(* Schneider Machine Expert - Basic project resolucao, file version 2.7.0.0 *)
(* ProjectInformations: Name=Novo projeto *)

HARDWARE
  Cpu 0: TM221M16R/G
  ModuleExtensionObject 0: TM3DQ16TK
  EthernetConfiguration: NetworkName=M221, IpAllocationMode=FixedAddress, IpAddress=0.0.0.0, SubnetMask=0.0.0.0
  SerialLineConfiguration: Baud=Baud19200, Parity=ParityEven, DataBits=DataBits8, StopBits=StopBits1, PhysicalMedium=PhysicalMediumRs485, TransmissionMode=TransmissionModeModbusRtu, SlaveId=1, Addressing=SlaveAddressing
  MastTask: UsePeriodScanMode=false, PeriodScan=100
  FastTask: Period=255
  CpuBehavior: StartingMode=StartAsPreviousState, AutoSaveRamOnEeprom=true, WatchdogPeriod=250

SYMBOLS  (address, symbol, comment, settings)
  %M0       SIG_IN_BOT_P1
  %M1       SIG_IN_BOT_P2
  %M2       SIG_IN_SEN_A
  %M3       SIG_IN_SEN_B
  %M4       SIG_IN_SEN_C
  %M5       SIG_IN_SEN_D1
  %M6       SIG_IN_SEN_D2
  %M10      SIG_E1_E2E3
  %M11      SIG_E2_E4
  %M13      SIG_E4_E6
  %M15      SIG_E6_E8
  %M17      SIG_E8_E10
  %M20      SIG_OUT_M1
  %M21      SIG_OUT_M1_INV
  %M22      SIG_OUT_M2
  %M23      SIG_OUT_M2_INV
  %M24      SIG_OUT_M3
  %M25      SIG_OUT_M3_INV
  %M26      SIG_OUT_M4
  %M27      SIG_OUT_M4_INV
  %M28      SIG_OUT_ATU_V1
  %M30      SIG_CAR_I_C
  %M31      SIG_CAR_II_C
  %M40      SIG_E10_E12
  %X1       E1
  %X2       E2
  %X3       E3
  %X4       E4
  %X5       E5
  %X6       E6
  %X7       E7
  %X8       E8
  %X9       E9
  %X10      E10
  %TM0      FT_E6_E8  [Preset=2, Base=OneSecond]
  %TM2      FT_E10_E12  [Preset=5, Base=OneSecond]
  %I0.0     IN_BOT_P1
  %I0.1     IN_BOT_P2
  %I0.2     IN_SEN_A
  %I0.3     IN_SEN_B
  %I0.4     IN_SEN_C
  %I0.5     IN_SEN_D1
  %I0.6     IN_SEN_D2
  %Q0.0     OUT_M1
  %Q0.1     OUT_M1_INV
  %Q0.2     OUT_M2
  %Q0.3     OUT_M2_INV
  %Q0.4     OUT_M3
  %Q0.5     OUT_M3_INV
  %Q0.6     OUT_M4
  %Q0.7     OUT_M4_INV
  %Q1.0     OUT_ATU_V1

GRAFCET Grafcet POU
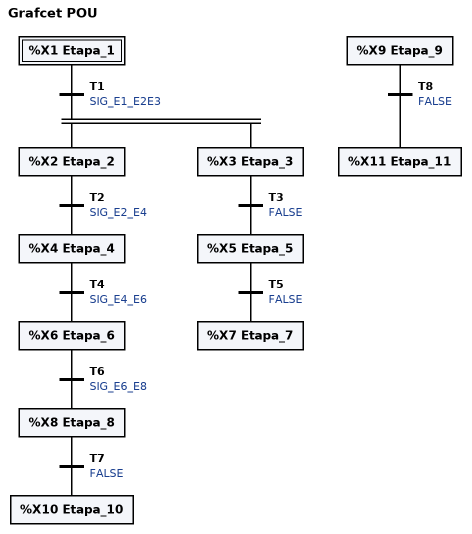
  INITIAL_STEP %X1  (* Etapa_1 *)
  STEP %X2  (* Etapa_2 *)
  STEP %X3  (* Etapa_3 *)
  STEP %X4  (* Etapa_4 *)
  STEP %X5  (* Etapa_5 *)
  STEP %X6  (* Etapa_6 *)
  STEP %X7  (* Etapa_7 *)
  STEP %X8  (* Etapa_8 *)
  STEP %X9  (* Etapa_9 *)
  STEP %X10  (* Etapa_10 *)
  STEP %X11  (* Etapa_11 *)
  TRANSITION T1 FROM %X1 TO %X2, %X3 := SIG_E1_E2E3;
  TRANSITION T2 FROM %X2 TO %X4 := SIG_E2_E4;
  TRANSITION T3 FROM %X3 TO %X5 := FALSE;
  TRANSITION T4 FROM %X4 TO %X6 := SIG_E4_E6;
  TRANSITION T5 FROM %X5 TO %X7 := FALSE;
  TRANSITION T6 FROM %X6 TO %X8 := SIG_E6_E8;
  TRANSITION T7 FROM %X8 TO %X10 := FALSE;
  TRANSITION T8 FROM %X9 TO %X11 := FALSE;

POU Entradas
  (* SectionNumber=0 *)

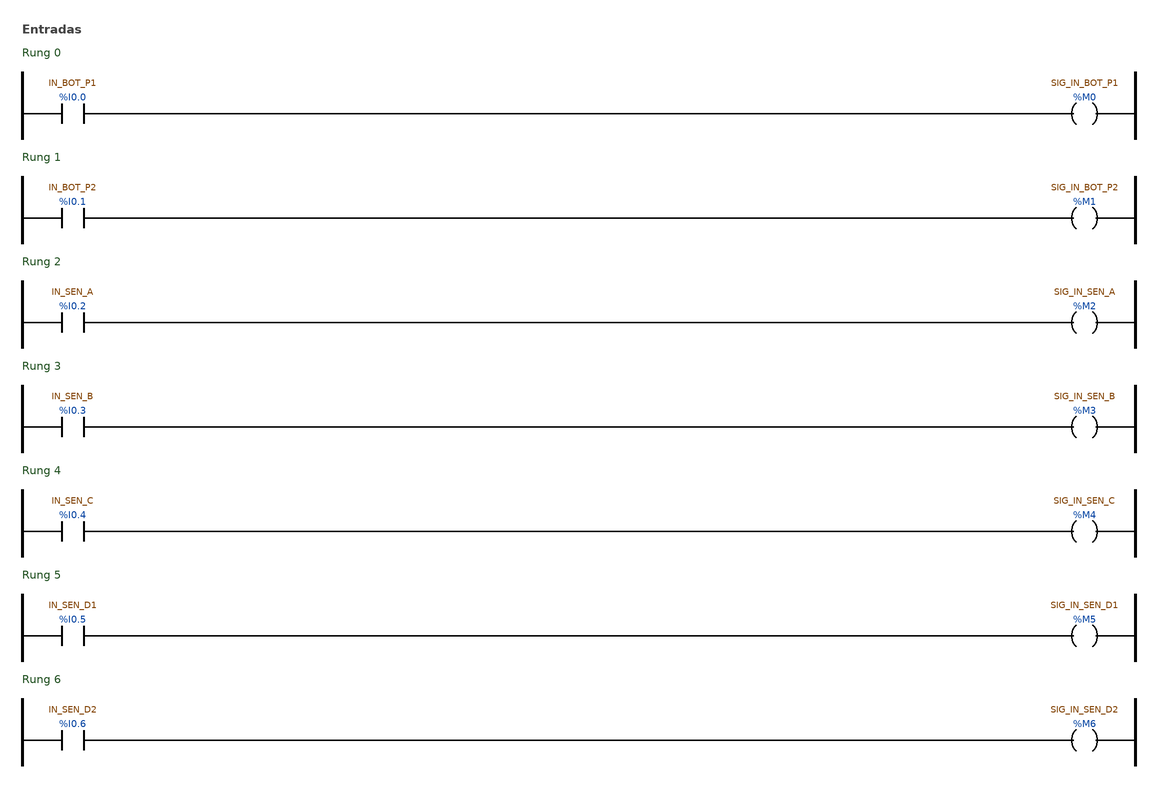

// Rung 0
  LD %I0.0                (* IN_BOT_P1 *)
  ST %M0                  (* SIG_IN_BOT_P1 *)
  // as ST:
  //   SIG_IN_BOT_P1 := IN_BOT_P1;

// Rung 1
  LD %I0.1                (* IN_BOT_P2 *)
  ST %M1                  (* SIG_IN_BOT_P2 *)
  // as ST:
  //   SIG_IN_BOT_P2 := IN_BOT_P2;

// Rung 2
  LD %I0.2                (* IN_SEN_A *)
  ST %M2                  (* SIG_IN_SEN_A *)
  // as ST:
  //   SIG_IN_SEN_A := IN_SEN_A;

// Rung 3
  LD %I0.3                (* IN_SEN_B *)
  ST %M3                  (* SIG_IN_SEN_B *)
  // as ST:
  //   SIG_IN_SEN_B := IN_SEN_B;

// Rung 4
  LD %I0.4                (* IN_SEN_C *)
  ST %M4                  (* SIG_IN_SEN_C *)
  // as ST:
  //   SIG_IN_SEN_C := IN_SEN_C;

// Rung 5
  LD %I0.5                (* IN_SEN_D1 *)
  ST %M5                  (* SIG_IN_SEN_D1 *)
  // as ST:
  //   SIG_IN_SEN_D1 := IN_SEN_D1;

// Rung 6
  LD %I0.6                (* IN_SEN_D2 *)
  ST %M6                  (* SIG_IN_SEN_D2 *)
  // as ST:
  //   SIG_IN_SEN_D2 := IN_SEN_D2;

TRANSITION T1 (%X1 -> %X2, %X3) 
  (* SectionNumber=0 *)

// Rung 7: E1_E2E3
  LD %M10                 (* SIG_E1_E2E3 *)
  ENDT
  // as ST:
  //   TRANSITION := SIG_E1_E2E3;

TRANSITION T2 (%X2 -> %X4) 
  (* SectionNumber=0 *)

// Rung 8: E2_E4
  LD %M11                 (* SIG_E2_E4 *)
  ENDT
  // as ST:
  //   TRANSITION := SIG_E2_E4;

TRANSITION T3 (%X3 -> %X5) 
  (* SectionNumber=0 *)

// Rung 9: E3_E5
  LD 0
  ENDT
  // as ST:
  //   TRANSITION := FALSE;

TRANSITION T4 (%X4 -> %X6) 
  (* SectionNumber=0 *)

// Rung 10: E4_E6
  LD %M13                 (* SIG_E4_E6 *)
  ENDT
  // as ST:
  //   TRANSITION := SIG_E4_E6;

TRANSITION T5 (%X5 -> %X7) 
  (* SectionNumber=0 *)

// Rung 11: Tr5
  LD 0
  ENDT
  // as ST:
  //   TRANSITION := FALSE;

TRANSITION T6 (%X6 -> %X8) 
  (* SectionNumber=0 *)

// Rung 12: E6_E8
  LD %M15                 (* SIG_E6_E8 *)
  ENDT
  // as ST:
  //   TRANSITION := SIG_E6_E8;

TRANSITION T7 (%X8 -> %X10) 
  (* SectionNumber=0 *)

// Rung 13: Tr7
  LD 0
  ENDT
  // as ST:
  //   TRANSITION := FALSE;

TRANSITION T8 (%X9 -> %X11) 
  (* SectionNumber=0 *)

// Rung 14: Tr8
  LD 0
  ENDT
  // as ST:
  //   TRANSITION := FALSE;

POU Lógicas
  (* SectionNumber=0 *)

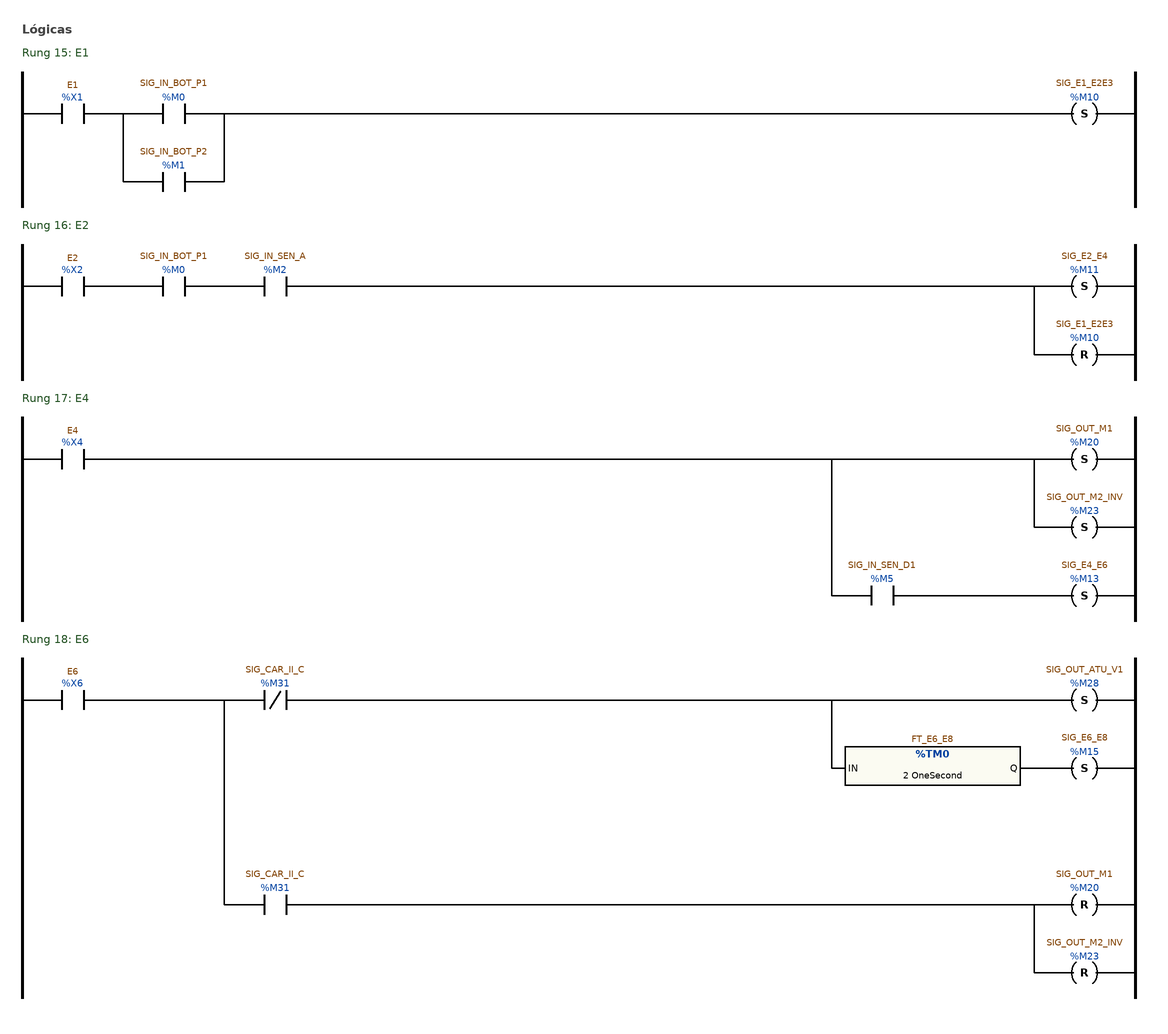

// Rung 15: E1
  LD %X1                  (* E1 *)
  AND( %M0                (* SIG_IN_BOT_P1 *)
  OR %M1                  (* SIG_IN_BOT_P2 *)
  )
  S %M10                  (* SIG_E1_E2E3 *)
  // as ST:
  //   IF E1 AND (SIG_IN_BOT_P1 OR SIG_IN_BOT_P2) THEN SIG_E1_E2E3 := TRUE; END_IF;

// Rung 16: E2
  LD %X2                  (* E2 *)
  AND %M0                 (* SIG_IN_BOT_P1 *)
  AND %M2                 (* SIG_IN_SEN_A *)
  S %M11                  (* SIG_E2_E4 *)
  R %M10                  (* SIG_E1_E2E3 *)
  // as ST:
  //   IF E2 AND SIG_IN_BOT_P1 AND SIG_IN_SEN_A THEN SIG_E2_E4 := TRUE; END_IF;
  //   IF E2 AND SIG_IN_BOT_P1 AND SIG_IN_SEN_A THEN SIG_E1_E2E3 := FALSE; END_IF;

// Rung 17: E4
  LD %X4                  (* E4 *)
  MPS
  S %M20                  (* SIG_OUT_M1 *)
  S %M23                  (* SIG_OUT_M2_INV *)
  MPP
  AND %M5                 (* SIG_IN_SEN_D1 *)
  S %M13                  (* SIG_E4_E6 *)
  // as ST:
  //   IF E4 THEN SIG_OUT_M1 := TRUE; END_IF;
  //   IF E4 THEN SIG_OUT_M2_INV := TRUE; END_IF;
  //   IF E4 AND SIG_IN_SEN_D1 THEN SIG_E4_E6 := TRUE; END_IF;

// Rung 18: E6
  LD 1
  MULTIFB
  LD 1
  AND %X6                 (* E6 *)
  ST %MW2009:X0
  LD %MW2009:X0
  ANDN %M31               (* SIG_CAR_II_C *)
  ST %MW2009:X1
  LD %MW2009:X1
  S %M28                  (* SIG_OUT_ATU_V1 *)
  BLK %TM0                (* FT_E6_E8 *)
  LD %MW2009:X1
  IN
  OUT_BLK
  LD Q
  S %M15                  (* SIG_E6_E8 *)
  END_BLK
  LD %MW2009:X0
  AND %M31                (* SIG_CAR_II_C *)
  R %M20                  (* SIG_OUT_M1 *)
  R %M23                  (* SIG_OUT_M2_INV *)
  MULTIFB
  // as ST:
  //   IF E6 AND NOT SIG_CAR_II_C THEN SIG_OUT_ATU_V1 := TRUE; END_IF;
  //   FT_E6_E8(IN := E6 AND NOT SIG_CAR_II_C);
  //   IF FT_E6_E8.Q THEN SIG_E6_E8 := TRUE; END_IF;
  //   IF E6 AND SIG_CAR_II_C THEN SIG_OUT_M1 := FALSE; END_IF;
  //   IF E6 AND SIG_CAR_II_C THEN SIG_OUT_M2_INV := FALSE; END_IF;

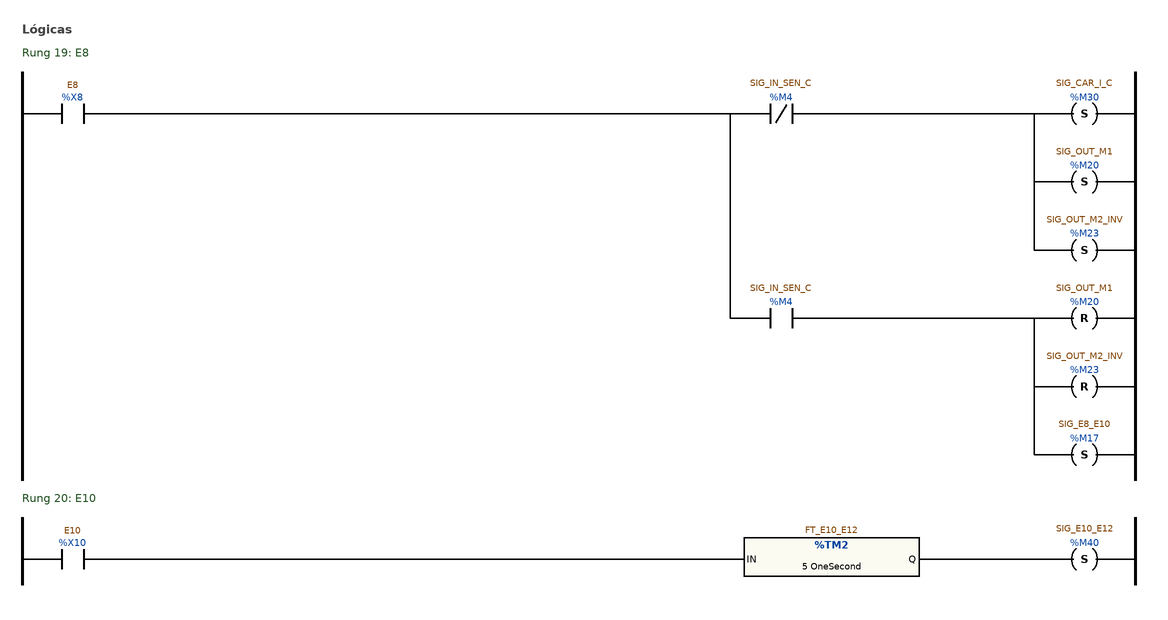

// Rung 19: E8
  LD %X8                  (* E8 *)
  MPS
  ANDN %M4                (* SIG_IN_SEN_C *)
  S %M30                  (* SIG_CAR_I_C *)
  S %M20                  (* SIG_OUT_M1 *)
  S %M23                  (* SIG_OUT_M2_INV *)
  MPP
  AND %M4                 (* SIG_IN_SEN_C *)
  R %M20                  (* SIG_OUT_M1 *)
  R %M23                  (* SIG_OUT_M2_INV *)
  S %M17                  (* SIG_E8_E10 *)
  // as ST:
  //   IF E8 AND NOT SIG_IN_SEN_C THEN SIG_CAR_I_C := TRUE; END_IF;
  //   IF E8 AND NOT SIG_IN_SEN_C THEN SIG_OUT_M1 := TRUE; END_IF;
  //   IF E8 AND NOT SIG_IN_SEN_C THEN SIG_OUT_M2_INV := TRUE; END_IF;
  //   IF E8 AND SIG_IN_SEN_C THEN SIG_OUT_M1 := FALSE; END_IF;
  //   IF E8 AND SIG_IN_SEN_C THEN SIG_OUT_M2_INV := FALSE; END_IF;
  //   IF E8 AND SIG_IN_SEN_C THEN SIG_E8_E10 := TRUE; END_IF;

// Rung 20: E10
  BLK %TM2                (* FT_E10_E12 *)
  LD %X10                 (* E10 *)
  IN
  OUT_BLK
  LD Q
  S %M40                  (* SIG_E10_E12 *)
  END_BLK
  // as ST:
  //   FT_E10_E12(IN := E10);
  //   IF FT_E10_E12.Q THEN SIG_E10_E12 := TRUE; END_IF;

POU Saídas
  (* SectionNumber=0 *)

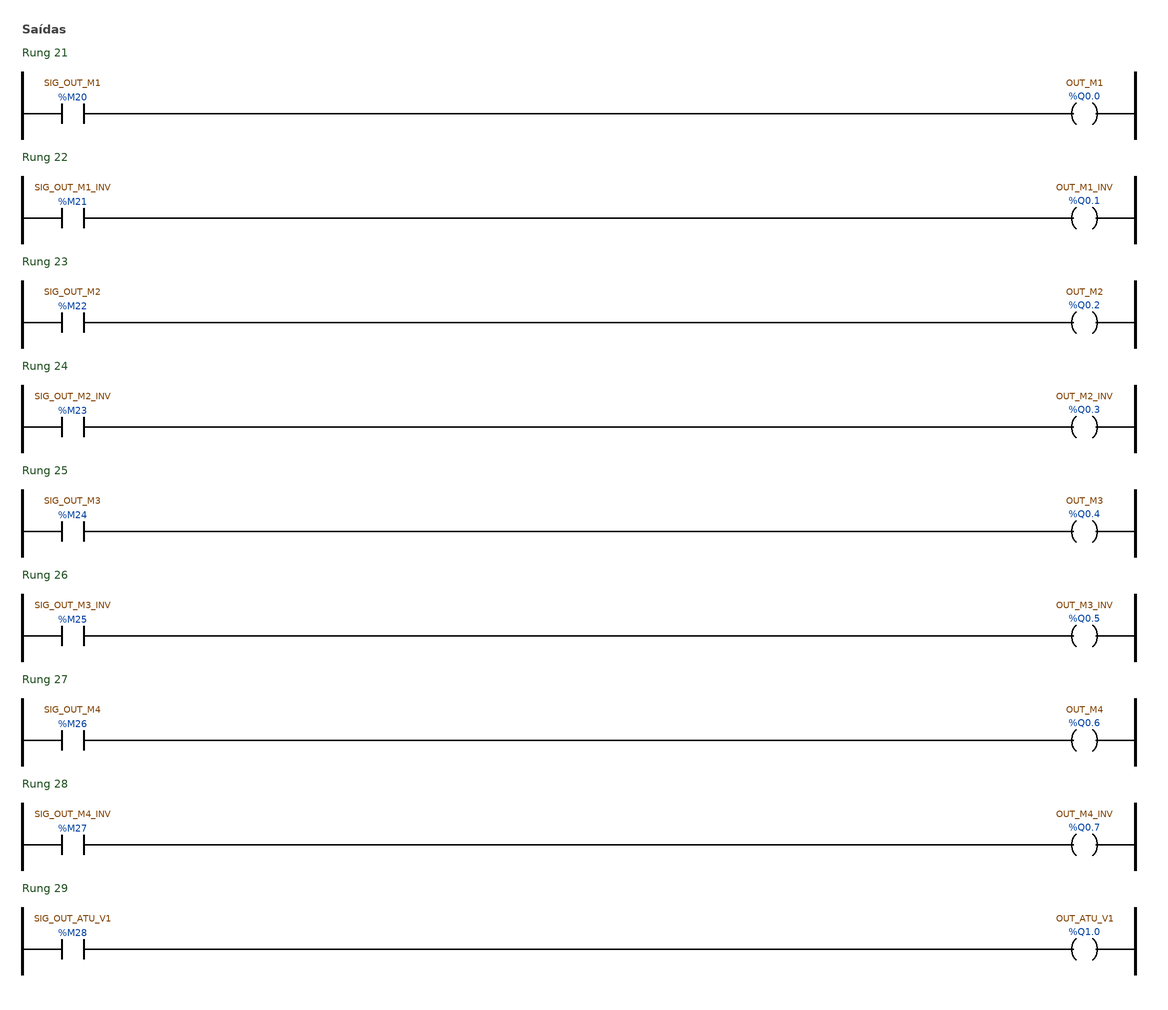

// Rung 21
  LD %M20                 (* SIG_OUT_M1 *)
  ST %Q0.0                (* OUT_M1 *)
  // as ST:
  //   OUT_M1 := SIG_OUT_M1;

// Rung 22
  LD %M21                 (* SIG_OUT_M1_INV *)
  ST %Q0.1                (* OUT_M1_INV *)
  // as ST:
  //   OUT_M1_INV := SIG_OUT_M1_INV;

// Rung 23
  LD %M22                 (* SIG_OUT_M2 *)
  ST %Q0.2                (* OUT_M2 *)
  // as ST:
  //   OUT_M2 := SIG_OUT_M2;

// Rung 24
  LD %M23                 (* SIG_OUT_M2_INV *)
  ST %Q0.3                (* OUT_M2_INV *)
  // as ST:
  //   OUT_M2_INV := SIG_OUT_M2_INV;

// Rung 25
  LD %M24                 (* SIG_OUT_M3 *)
  ST %Q0.4                (* OUT_M3 *)
  // as ST:
  //   OUT_M3 := SIG_OUT_M3;

// Rung 26
  LD %M25                 (* SIG_OUT_M3_INV *)
  ST %Q0.5                (* OUT_M3_INV *)
  // as ST:
  //   OUT_M3_INV := SIG_OUT_M3_INV;

// Rung 27
  LD %M26                 (* SIG_OUT_M4 *)
  ST %Q0.6                (* OUT_M4 *)
  // as ST:
  //   OUT_M4 := SIG_OUT_M4;

// Rung 28
  LD %M27                 (* SIG_OUT_M4_INV *)
  ST %Q0.7                (* OUT_M4_INV *)
  // as ST:
  //   OUT_M4_INV := SIG_OUT_M4_INV;

// Rung 29
  LD %M28                 (* SIG_OUT_ATU_V1 *)
  ST %Q1.0                (* OUT_ATU_V1 *)
  // as ST:
  //   OUT_ATU_V1 := SIG_OUT_ATU_V1;
